(* Logix 5000 project; controller Sucrose_Main Emulate 5570 rev 20.12; software revision 20.01; part 27 of 30 *)
(* tags used below, declared in another part *)
   AI_E23_0 : REAL[8];   // Analog Input EN2T_FLX 192.168.1.23
   AI_E23_1 : REAL[8];   // Analog Input EN2T_FLX 192.168.1.23
   Alarm_ACK_Master_Timer : TIMER;
   DI_E23_3 : ALIAS FOR FLX_E23:3:I;   // Discrete Input EN2T_FLX 192.168.1.23
   DO_E24_2 : ALIAS FOR FLX_E24:2:O;   // Discrete Output EN2T_FLX 192.168.1.24
   DO_E24_3 : ALIAS FOR FLX_E24:3:O;   // Discrete Output EN2T_FLX 192.168.1.24
   DO_E24_4 : ALIAS FOR FLX_E24:4:O;   // Discrete Output EN2T_FLX 192.168.1.24
   FV740301_AOI : QSI_Flow_Valve;   // FV-74-03-01 STEAM SIP SUPPLY VALVE
   FV751401_AOI : QSI_Flow_Valve;   // FV-75-14-01 CONDENSATE TANK BLANKETING STEAM TRAP ISOLATION VALVE
   FV920301_AOI : QSI_Flow_Valve;   // FV-92-03-01 INSTRUMENT AIR HEATER ISOLATION VALVE
   HTR920301_AOI : QSI_Discrete_Device;   // HTR-92-03-01 COMPRESSED AIR TANK AIR BLANKETING HEATER
   PIT_93_01_01_HIGH_PRESS : DINT;
   PIT_93_01_01_LOW_PRESS : DINT;
   PIT_93_02_01_HIGH_PRESS : DINT;
   PIT_93_02_01_LOW_PRESS : DINT;
   PIT_93_03_01_HIGH_PRESS : DINT;
   PIT_93_03_01_LOW_PRESS : DINT;
   Rung_Comment : BOOL;
   Sucrose_MM_Enable : BOOL;
   SucroseCIP_TK230101_REMOTE : CIP_REMOTE;
   SucroseCIP_TK230201_REMOTE : CIP_REMOTE;
   SucroseCIP_TK230301_REMOTE : CIP_REMOTE;
   SucroseDischarge : Area_Program;
   SucroseTanks : Area_Program;
   TK_23_01_01_HIGH_LEVEL : DINT;
   TK_23_01_01_HIGH_TEMP : DINT;
   TK_23_01_01_LOW_LEVEL : DINT;
   TK_23_01_01_LOW_TEMP : DINT;
   TK_23_01_01_NO_PRESS_ALARM : BOOL;
   TK_23_01_01_NO_TEMP_ALARM : BOOL;
   TK_23_01_01_TEMP_LEVEL : DINT;
   TK_23_02_01_HIGH_LEVEL : DINT;
   TK_23_02_01_HIGH_TEMP : DINT;
   TK_23_02_01_LOW_LEVEL : DINT;
   TK_23_02_01_LOW_TEMP : DINT;
   TK_23_02_01_NO_PRESS_ALARM : BOOL;
   TK_23_02_01_NO_TEMP_ALARM : BOOL;
   TK_23_02_01_TEMP_LEVEL : DINT;
   TK_23_03_01_HIGH_LEVEL : DINT;
   TK_23_03_01_HIGH_TEMP : DINT;
   TK_23_03_01_LOW_LEVEL : DINT;
   TK_23_03_01_LOW_TEMP : DINT;
   TK_23_03_01_NO_PRESS_ALARM : BOOL;
   TK_23_03_01_NO_TEMP_ALARM : BOOL;
   TK_23_03_01_TEMP_LEVEL : DINT;
(* Steam_AirArea_AutoLogic, continued *)

ROUTINE Enable_Logic   (* ladder *)
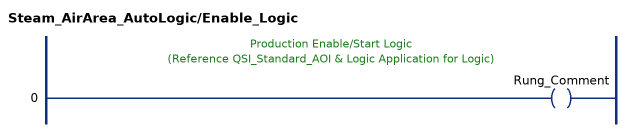
   // Production Enable/Start Logic
   // (Reference QSI_Standard_AOI & Logic Application for Logic)
   0: OTE(Rung_Comment);
END_ROUTINE

ROUTINE MainRoutine   (* ladder *)
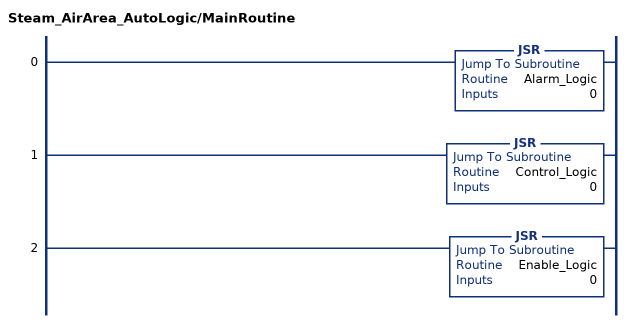
   0: JSR(Alarm_Logic,0);
   1: JSR(Control_Logic,0);
   2: JSR(Enable_Logic,0);
END_ROUTINE
END_PROGRAM

PROGRAM Steam_AirArea_EN2T_IO_Discrete_DO_E24_2   (* main routine MainRoutine *)

ROUTINE _12_HTR920301   (* ladder *)
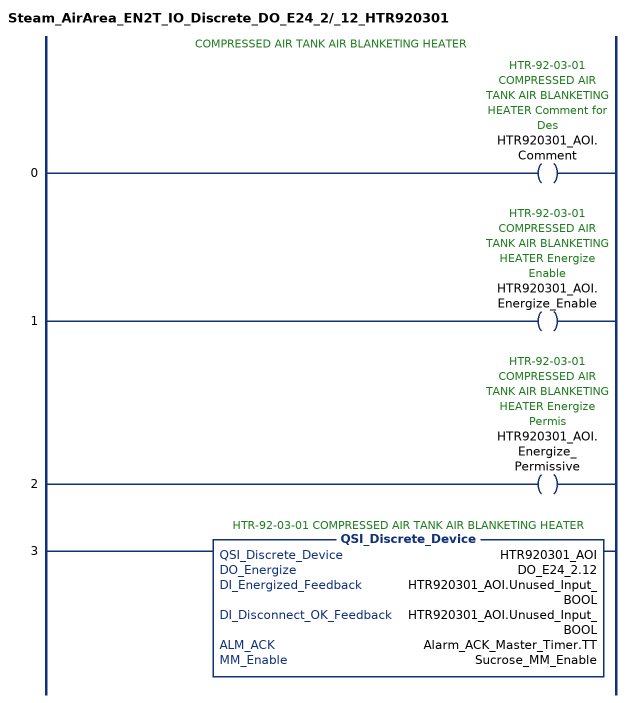
   // COMPRESSED AIR TANK AIR BLANKETING HEATER
   0: OTE(HTR920301_AOI.Comment);
   1: OTE(HTR920301_AOI.Energize_Enable);
   2: OTE(HTR920301_AOI.Energize_Permissive);
   3: QSI_Discrete_Device(HTR920301_AOI,DO_E24_2.12,HTR920301_AOI.Unused_Input_BOOL,HTR920301_AOI.Unused_Input_BOOL,Alarm_ACK_Master_Timer.TT,Sucrose_MM_Enable);
END_ROUTINE

ROUTINE MainRoutine   (* ladder *)
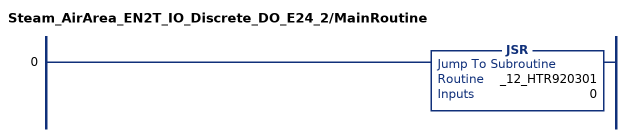
   0: JSR(_12_HTR920301,0);
END_ROUTINE
END_PROGRAM

PROGRAM Steam_AirArea_EN2T_IO_Discrete_DO_E24_3   (* main routine MainRoutine *)

ROUTINE _14_FV751401   (* ladder *)
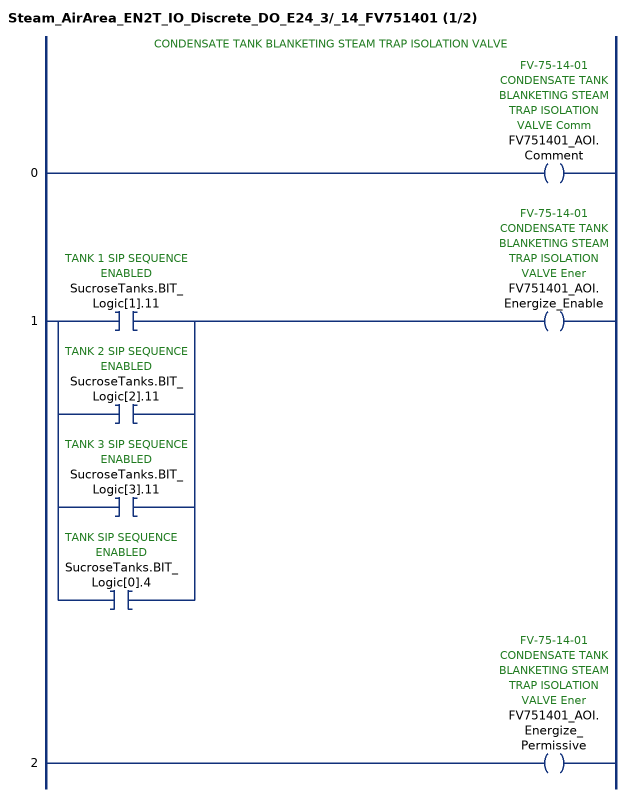
   // CONDENSATE TANK BLANKETING STEAM TRAP ISOLATION VALVE
   0: OTE(FV751401_AOI.Comment);
   1: [XIC(SucroseTanks.BIT_Logic[1].11) ,XIC(SucroseTanks.BIT_Logic[2].11) ,XIC(SucroseTanks.BIT_Logic[3].11) ,XIC(SucroseTanks.BIT_Logic[0].4) ]OTE(FV751401_AOI.Energize_Enable);
   2: OTE(FV751401_AOI.Energize_Permissive);
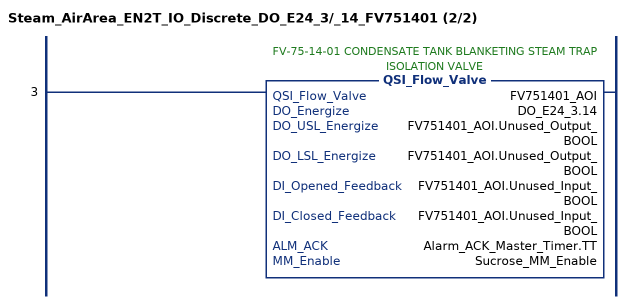
   3: QSI_Flow_Valve(FV751401_AOI,DO_E24_3.14,FV751401_AOI.Unused_Output_BOOL,FV751401_AOI.Unused_Output_BOOL,FV751401_AOI.Unused_Input_BOOL,FV751401_AOI.Unused_Input_BOOL,Alarm_ACK_Master_Timer.TT,Sucrose_MM_Enable);
END_ROUTINE

ROUTINE _15_FV920301   (* ladder *)
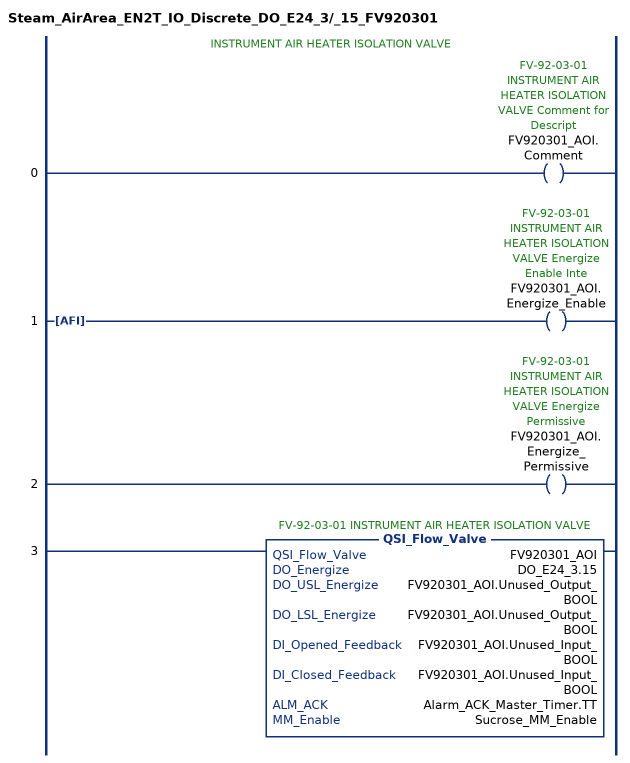
   // INSTRUMENT AIR HEATER ISOLATION VALVE
   0: OTE(FV920301_AOI.Comment);
   1: AFI()OTE(FV920301_AOI.Energize_Enable);
   2: OTE(FV920301_AOI.Energize_Permissive);
   3: QSI_Flow_Valve(FV920301_AOI,DO_E24_3.15,FV920301_AOI.Unused_Output_BOOL,FV920301_AOI.Unused_Output_BOOL,FV920301_AOI.Unused_Input_BOOL,FV920301_AOI.Unused_Input_BOOL,Alarm_ACK_Master_Timer.TT,Sucrose_MM_Enable);
END_ROUTINE

ROUTINE MainRoutine   (* ladder *)
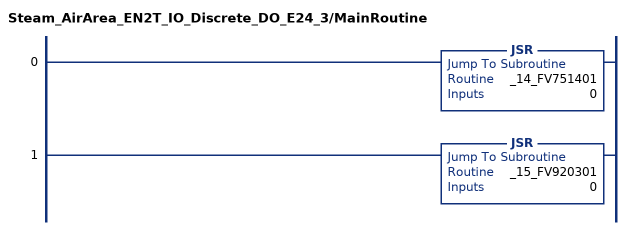
   0: JSR(_14_FV751401,0);
   1: JSR(_15_FV920301,0);
END_ROUTINE
END_PROGRAM

PROGRAM Steam_AirArea_EN2T_IO_Discrete_DO_E24_4   (* main routine MainRoutine *)

ROUTINE _00_FV740301   (* ladder *)
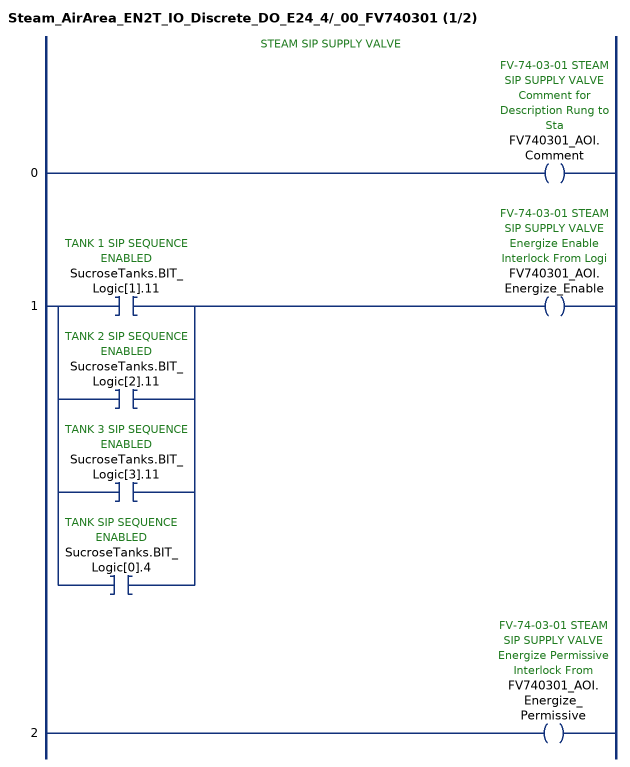
   // STEAM SIP SUPPLY VALVE
   0: OTE(FV740301_AOI.Comment);
   1: [XIC(SucroseTanks.BIT_Logic[1].11) ,XIC(SucroseTanks.BIT_Logic[2].11) ,XIC(SucroseTanks.BIT_Logic[3].11) ,XIC(SucroseTanks.BIT_Logic[0].4) ]OTE(FV740301_AOI.Energize_Enable);
   2: OTE(FV740301_AOI.Energize_Permissive);
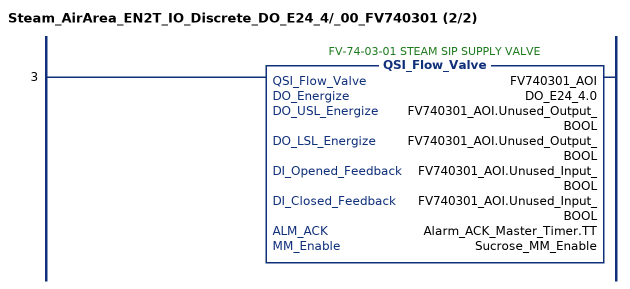
   3: QSI_Flow_Valve(FV740301_AOI,DO_E24_4.0,FV740301_AOI.Unused_Output_BOOL,FV740301_AOI.Unused_Output_BOOL,FV740301_AOI.Unused_Input_BOOL,FV740301_AOI.Unused_Input_BOOL,Alarm_ACK_Master_Timer.TT,Sucrose_MM_Enable);
END_ROUTINE

ROUTINE MainRoutine   (* ladder *)
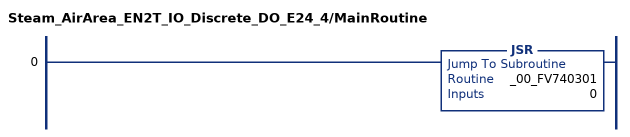
   0: JSR(_00_FV740301,0);
END_ROUTINE
END_PROGRAM

PROGRAM TanksArea_AutoLogic   (* main routine MainRoutine *)

ROUTINE Alarm_Logic   (* ladder *)
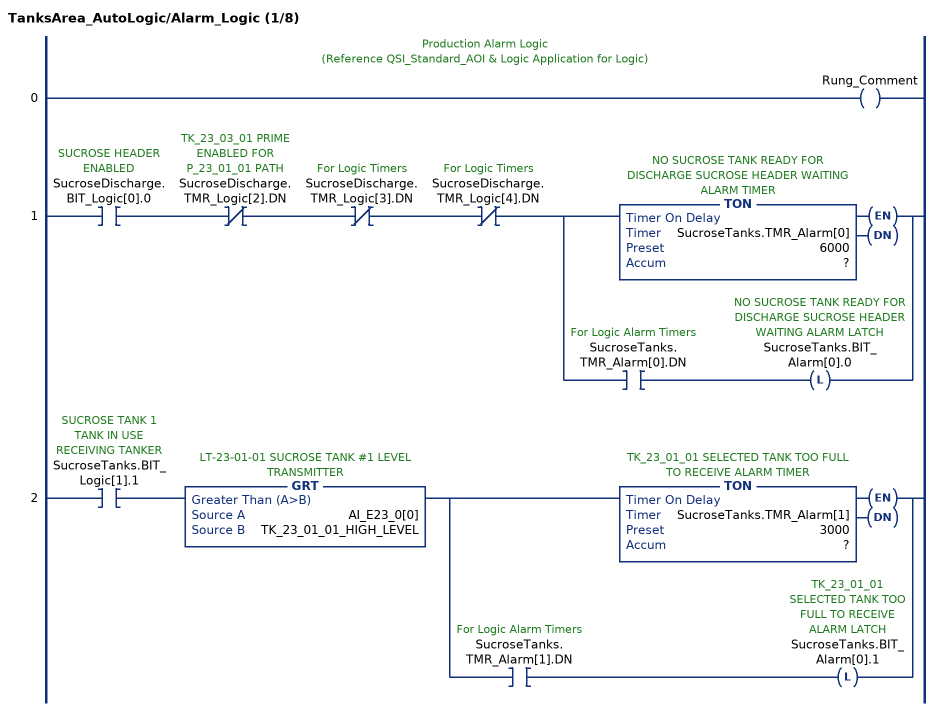
   // Production Alarm Logic
   // (Reference QSI_Standard_AOI & Logic Application for Logic)
   0: OTE(Rung_Comment);
   1: XIC(SucroseDischarge.BIT_Logic[0].0)XIO(SucroseDischarge.TMR_Logic[2].DN)XIO(SucroseDischarge.TMR_Logic[3].DN)XIO(SucroseDischarge.TMR_Logic[4].DN)[TON(SucroseTanks.TMR_Alarm[0],?,?) ,XIC(SucroseTanks.TMR_Alarm[0].DN) OTL(SucroseTanks.BIT_Alarm[0].0) ];
   2: XIC(SucroseTanks.BIT_Logic[1].1)GRT(AI_E23_0[0],TK_23_01_01_HIGH_LEVEL)[TON(SucroseTanks.TMR_Alarm[1],?,?) ,XIC(SucroseTanks.TMR_Alarm[1].DN) OTL(SucroseTanks.BIT_Alarm[0].1) ];
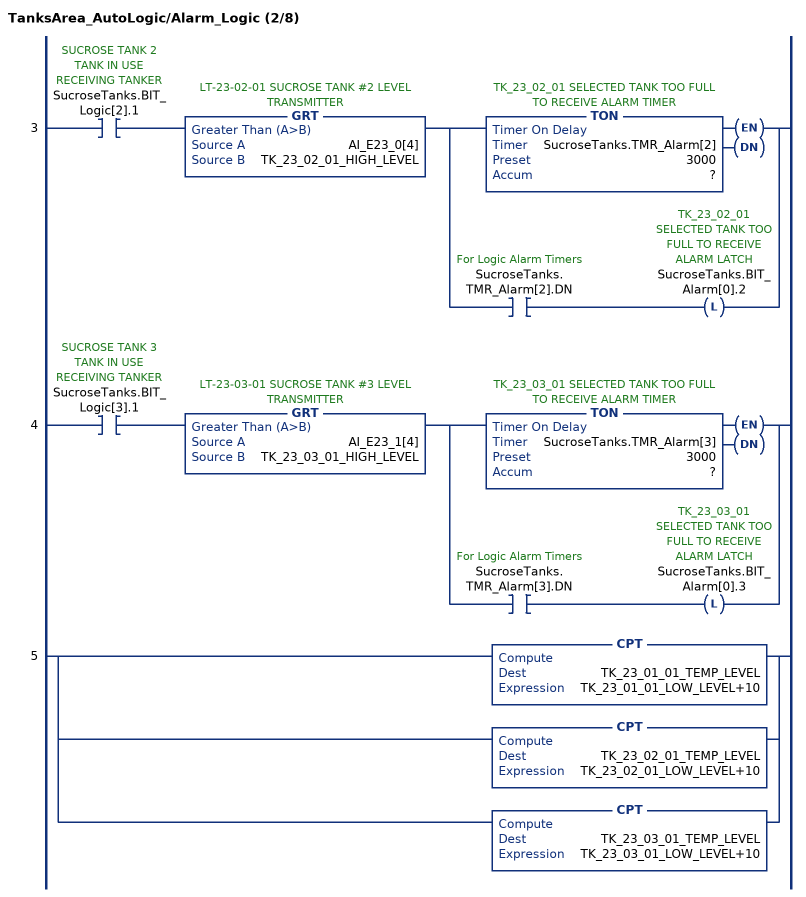
   3: XIC(SucroseTanks.BIT_Logic[2].1)GRT(AI_E23_0[4],TK_23_02_01_HIGH_LEVEL)[TON(SucroseTanks.TMR_Alarm[2],?,?) ,XIC(SucroseTanks.TMR_Alarm[2].DN) OTL(SucroseTanks.BIT_Alarm[0].2) ];
   4: XIC(SucroseTanks.BIT_Logic[3].1)GRT(AI_E23_1[4],TK_23_03_01_HIGH_LEVEL)[TON(SucroseTanks.TMR_Alarm[3],?,?) ,XIC(SucroseTanks.TMR_Alarm[3].DN) OTL(SucroseTanks.BIT_Alarm[0].3) ];
   5: [CPT(TK_23_01_01_TEMP_LEVEL,TK_23_01_01_LOW_LEVEL+10) ,CPT(TK_23_02_01_TEMP_LEVEL,TK_23_02_01_LOW_LEVEL+10) ,CPT(TK_23_03_01_TEMP_LEVEL,TK_23_03_01_LOW_LEVEL+10) ];
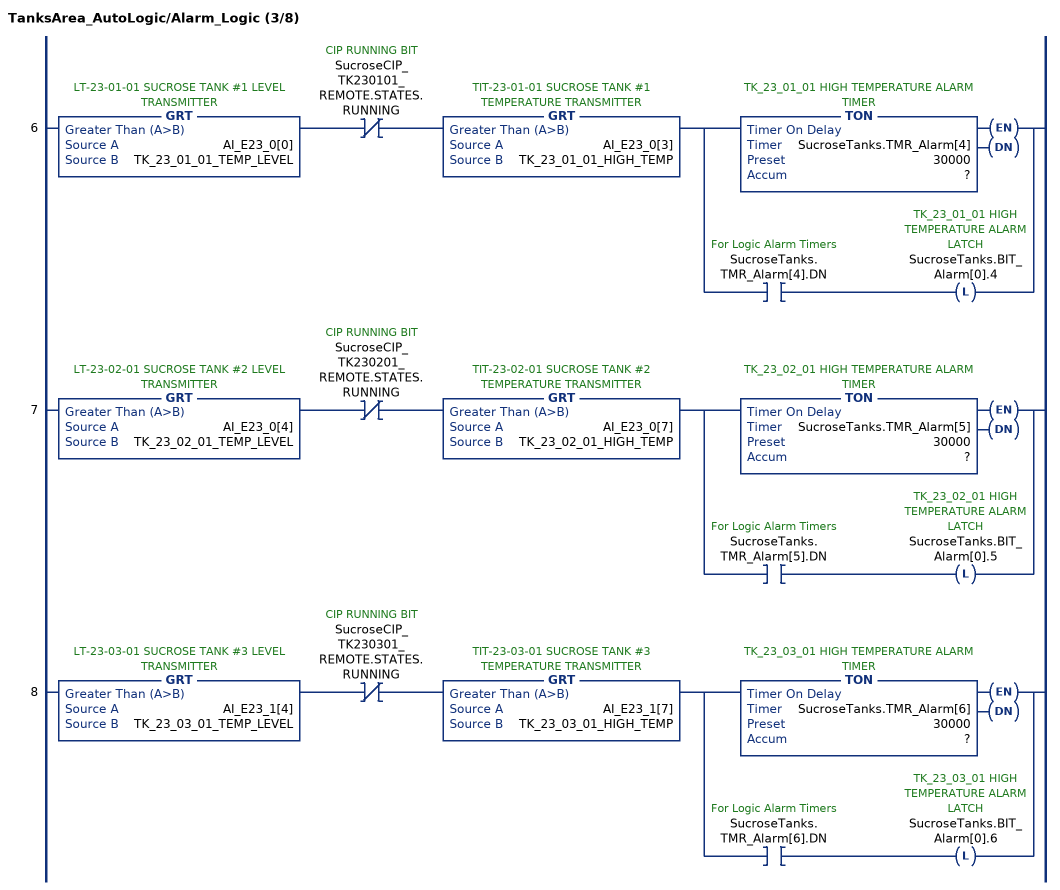
   6: GRT(AI_E23_0[0],TK_23_01_01_TEMP_LEVEL)XIO(SucroseCIP_TK230101_REMOTE.STATES.RUNNING)GRT(AI_E23_0[3],TK_23_01_01_HIGH_TEMP)[TON(SucroseTanks.TMR_Alarm[4],?,?) ,XIC(SucroseTanks.TMR_Alarm[4].DN) OTL(SucroseTanks.BIT_Alarm[0].4) ];
   7: GRT(AI_E23_0[4],TK_23_02_01_TEMP_LEVEL)XIO(SucroseCIP_TK230201_REMOTE.STATES.RUNNING)GRT(AI_E23_0[7],TK_23_02_01_HIGH_TEMP)[TON(SucroseTanks.TMR_Alarm[5],?,?) ,XIC(SucroseTanks.TMR_Alarm[5].DN) OTL(SucroseTanks.BIT_Alarm[0].5) ];
   8: GRT(AI_E23_1[4],TK_23_03_01_TEMP_LEVEL)XIO(SucroseCIP_TK230301_REMOTE.STATES.RUNNING)GRT(AI_E23_1[7],TK_23_03_01_HIGH_TEMP)[TON(SucroseTanks.TMR_Alarm[6],?,?) ,XIC(SucroseTanks.TMR_Alarm[6].DN) OTL(SucroseTanks.BIT_Alarm[0].6) ];
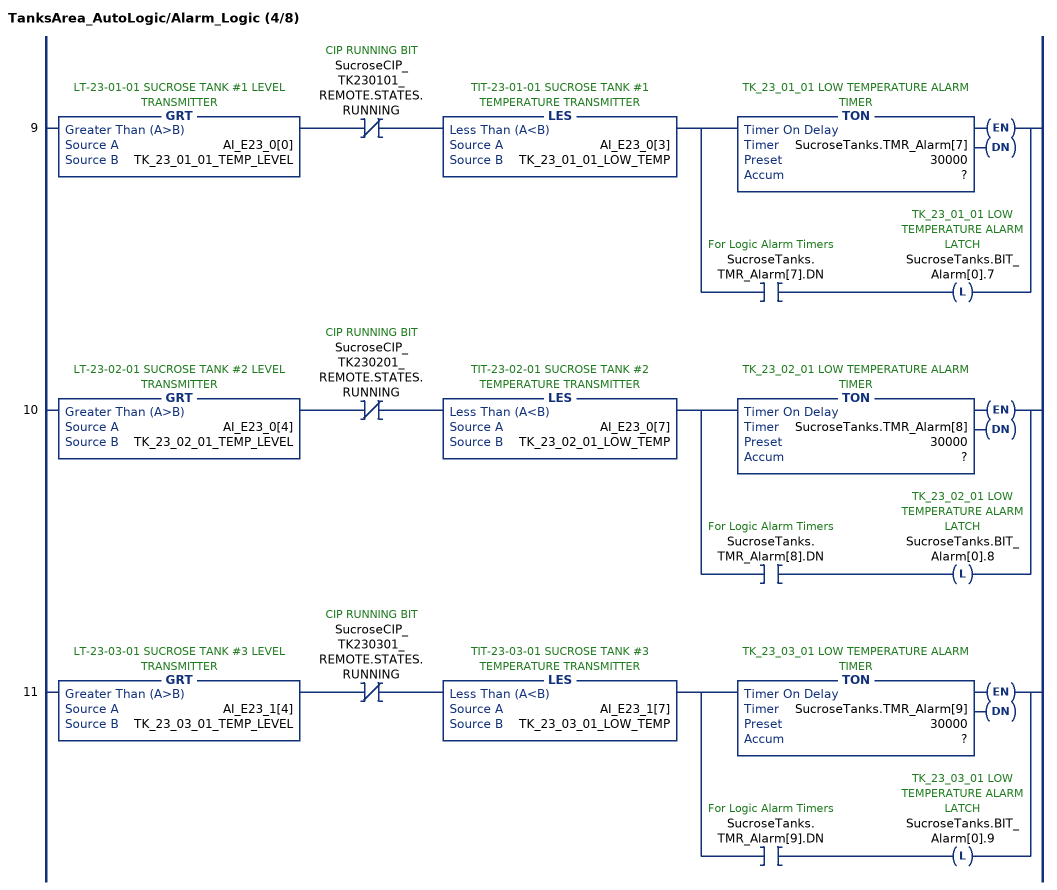
   9: GRT(AI_E23_0[0],TK_23_01_01_TEMP_LEVEL)XIO(SucroseCIP_TK230101_REMOTE.STATES.RUNNING)LES(AI_E23_0[3],TK_23_01_01_LOW_TEMP)[TON(SucroseTanks.TMR_Alarm[7],?,?) ,XIC(SucroseTanks.TMR_Alarm[7].DN) OTL(SucroseTanks.BIT_Alarm[0].7) ];
   10: GRT(AI_E23_0[4],TK_23_02_01_TEMP_LEVEL)XIO(SucroseCIP_TK230201_REMOTE.STATES.RUNNING)LES(AI_E23_0[7],TK_23_02_01_LOW_TEMP)[TON(SucroseTanks.TMR_Alarm[8],?,?) ,XIC(SucroseTanks.TMR_Alarm[8].DN) OTL(SucroseTanks.BIT_Alarm[0].8) ];
   11: GRT(AI_E23_1[4],TK_23_03_01_TEMP_LEVEL)XIO(SucroseCIP_TK230301_REMOTE.STATES.RUNNING)LES(AI_E23_1[7],TK_23_03_01_LOW_TEMP)[TON(SucroseTanks.TMR_Alarm[9],?,?) ,XIC(SucroseTanks.TMR_Alarm[9].DN) OTL(SucroseTanks.BIT_Alarm[0].9) ];
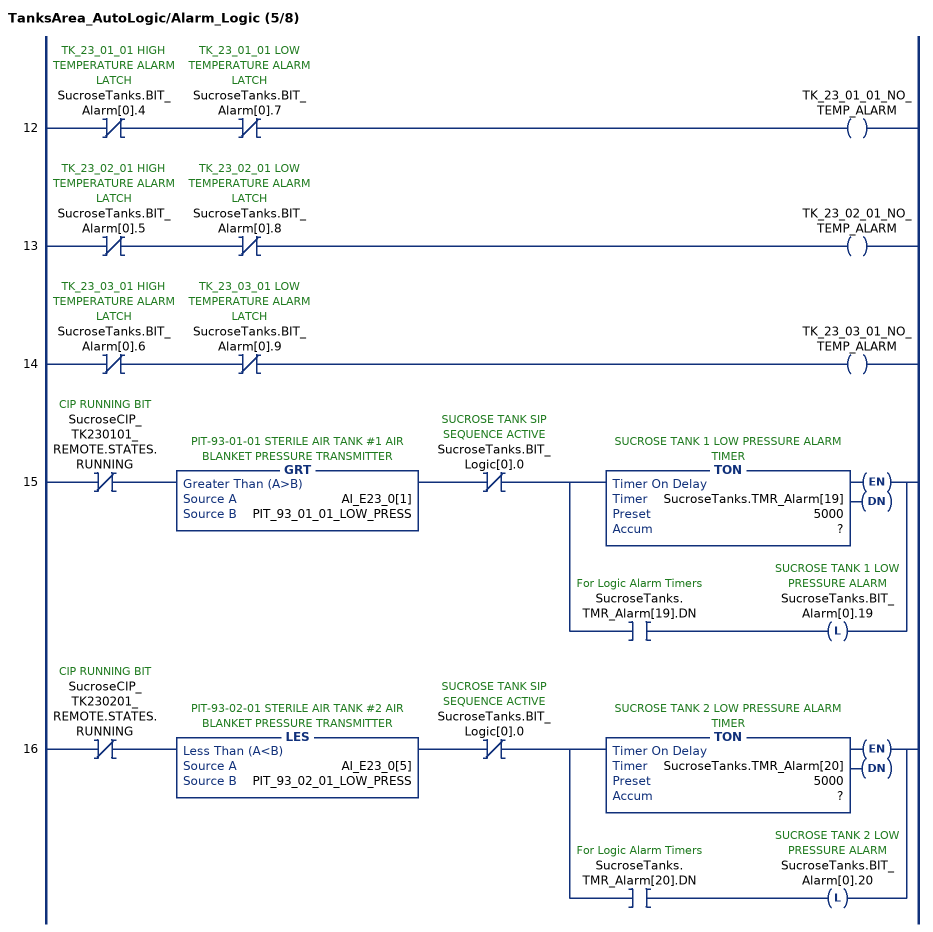
   12: XIO(SucroseTanks.BIT_Alarm[0].4)XIO(SucroseTanks.BIT_Alarm[0].7)OTE(TK_23_01_01_NO_TEMP_ALARM);
   13: XIO(SucroseTanks.BIT_Alarm[0].5)XIO(SucroseTanks.BIT_Alarm[0].8)OTE(TK_23_02_01_NO_TEMP_ALARM);
   14: XIO(SucroseTanks.BIT_Alarm[0].6)XIO(SucroseTanks.BIT_Alarm[0].9)OTE(TK_23_03_01_NO_TEMP_ALARM);
   15: XIO(SucroseCIP_TK230101_REMOTE.STATES.RUNNING)GRT(AI_E23_0[1],PIT_93_01_01_LOW_PRESS)XIO(SucroseTanks.BIT_Logic[0].0)[TON(SucroseTanks.TMR_Alarm[19],?,?) ,XIC(SucroseTanks.TMR_Alarm[19].DN) OTL(SucroseTanks.BIT_Alarm[0].19) ];
   16: XIO(SucroseCIP_TK230201_REMOTE.STATES.RUNNING)LES(AI_E23_0[5],PIT_93_02_01_LOW_PRESS)XIO(SucroseTanks.BIT_Logic[0].0)[TON(SucroseTanks.TMR_Alarm[20],?,?) ,XIC(SucroseTanks.TMR_Alarm[20].DN) OTL(SucroseTanks.BIT_Alarm[0].20) ];
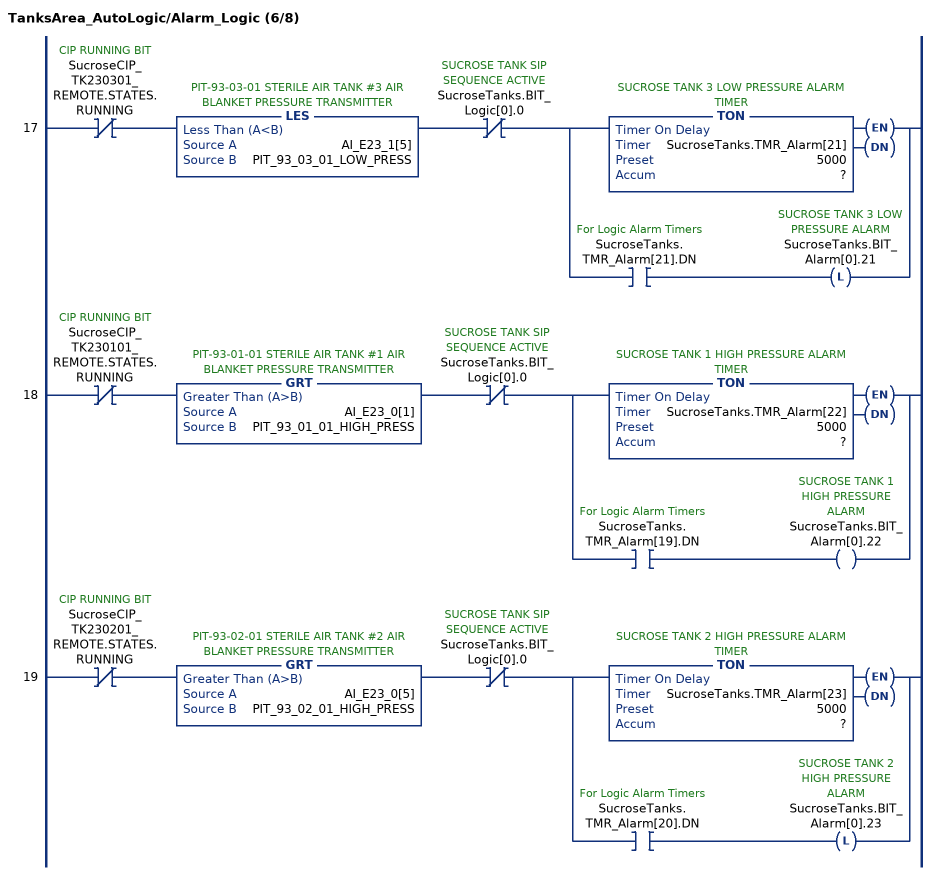
   17: XIO(SucroseCIP_TK230301_REMOTE.STATES.RUNNING)LES(AI_E23_1[5],PIT_93_03_01_LOW_PRESS)XIO(SucroseTanks.BIT_Logic[0].0)[TON(SucroseTanks.TMR_Alarm[21],?,?) ,XIC(SucroseTanks.TMR_Alarm[21].DN) OTL(SucroseTanks.BIT_Alarm[0].21) ];
   18: XIO(SucroseCIP_TK230101_REMOTE.STATES.RUNNING)GRT(AI_E23_0[1],PIT_93_01_01_HIGH_PRESS)XIO(SucroseTanks.BIT_Logic[0].0)[TON(SucroseTanks.TMR_Alarm[22],?,?) ,XIC(SucroseTanks.TMR_Alarm[19].DN) OTE(SucroseTanks.BIT_Alarm[0].22) ];
   19: XIO(SucroseCIP_TK230201_REMOTE.STATES.RUNNING)GRT(AI_E23_0[5],PIT_93_02_01_HIGH_PRESS)XIO(SucroseTanks.BIT_Logic[0].0)[TON(SucroseTanks.TMR_Alarm[23],?,?) ,XIC(SucroseTanks.TMR_Alarm[20].DN) OTL(SucroseTanks.BIT_Alarm[0].23) ];
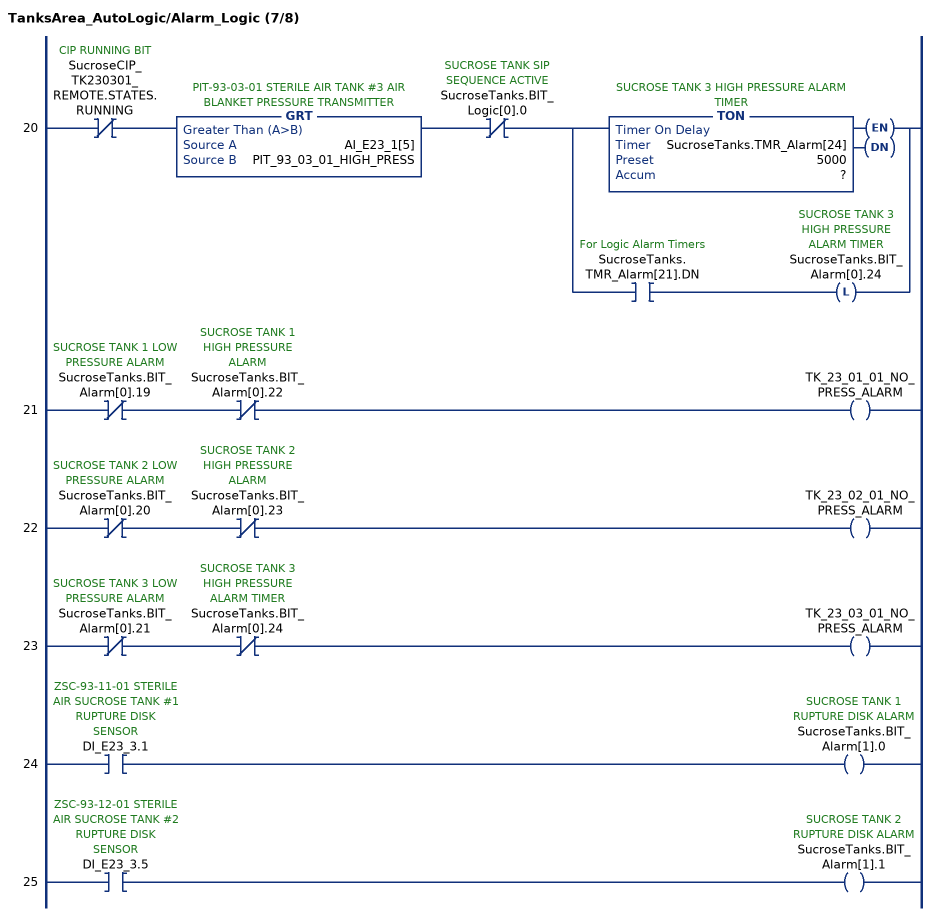
   20: XIO(SucroseCIP_TK230301_REMOTE.STATES.RUNNING)GRT(AI_E23_1[5],PIT_93_03_01_HIGH_PRESS)XIO(SucroseTanks.BIT_Logic[0].0)[TON(SucroseTanks.TMR_Alarm[24],?,?) ,XIC(SucroseTanks.TMR_Alarm[21].DN) OTL(SucroseTanks.BIT_Alarm[0].24) ];
   21: XIO(SucroseTanks.BIT_Alarm[0].19)XIO(SucroseTanks.BIT_Alarm[0].22)OTE(TK_23_01_01_NO_PRESS_ALARM);
   22: XIO(SucroseTanks.BIT_Alarm[0].20)XIO(SucroseTanks.BIT_Alarm[0].23)OTE(TK_23_02_01_NO_PRESS_ALARM);
   23: XIO(SucroseTanks.BIT_Alarm[0].21)XIO(SucroseTanks.BIT_Alarm[0].24)OTE(TK_23_03_01_NO_PRESS_ALARM);
   24: XIC(DI_E23_3.1)OTE(SucroseTanks.BIT_Alarm[1].0);
   25: XIC(DI_E23_3.5)OTE(SucroseTanks.BIT_Alarm[1].1);
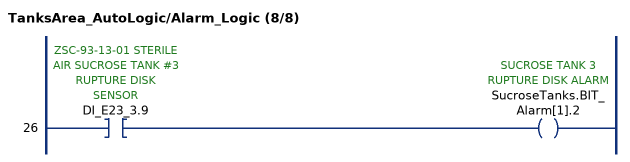
   26: XIC(DI_E23_3.9)OTE(SucroseTanks.BIT_Alarm[1].2);
END_ROUTINE
